TYPE ST_EL2809_B :
STRUCT
	//--------------------------------------------------------------------------------------------------------
	sTerminalName                                           :   STRING(200):= 'EL2809 | 16-Channel Digital Output';
	//=============================================================================================================
	// TERMINAL - EL2809	16-Channel Digital Output Terminal	 (Term 9)
	qExtendProcessCylinder2					AT %Q*			: 	BOOL;	// EL2809 channel 1
	qRetractProcessCylinder2				AT %Q* 			: 	BOOL;	// EL2809 channel 2
	qPartHolder2		             		AT %Q*	 		: 	BOOL;	// EL2809 channel 3 			
	iEL2809_B_Ch4			      			AT %Q*	 		: 	BOOL;	// EL2809 channel 4 
	qExtendVacuumCylinder2			  		AT %Q*	 		: 	BOOL;	// EL2809 channel 5
	qRetractVacuumCylinder2		 			AT %Q*	 		: 	BOOL;	// EL2809 channel 6 	
	iEL2809_B_Ch7         		    		AT %Q*			: 	BOOL;	// EL2809 channel 7	
	iEL2809_B_Ch8							AT %Q*	 		: 	BOOL;	// EL2809 channel 8	
	iEL2809_B_Ch9                 			AT %Q*          :   BOOL;   // EL2809 channel 9
	iEL2809_B_Ch10            				AT %Q*          :   BOOL;   // EL2809 channel 10   	
	iEL2809_B_Ch11    						AT %Q*	 		: 	BOOL;	// EL2809 channel 11	
	iEL2809_B_Ch12  						AT %Q*	 		: 	BOOL;	// EL2809 channel 12 
    iEL2809_B_Ch13			        		AT %Q*	 		: 	BOOL;	// EL2809 channel 13 
	iEL2809_B_Ch14               			AT %Q*	 		: 	BOOL;	// EL2809 channel 14 
	iEL2809_B_Ch15							AT %Q*	 		: 	BOOL;	// EL2809 channel 15 
    iEL2809_B_Ch16 	        				AT %Q*	 		: 	BOOL;	// EL2809 channel 16
	
	stTerminalInfo											: 	ST_Terminal_Info;

	
END_STRUCT
END_TYPE

(* stored: Version 1.1.0.1, ProductVersion 3.1.4026.18
   DUT ST_EL2809_B: Id {a57da4c4-94c5-4b4c-84af-e8a4ba5a5add} *)
